TEXTLIST tlPML_Modes
  0 = 'PMLUnitMode_Invalid'
  1 = 'PMLUnitMode_Production'
  2 = 'PMLUnitMode_Maintenance'
  3 = 'PMLUnitMode_Manual'
   = ''
END_TEXTLIST

(* stored: Version 1.1.0.1, ProductVersion 3.1.4024.11
   TextList tlPML_Modes: Id {79718370-c230-4441-9a2b-44dfe1194bec} *)
